FUNCTION F_TemperatureMethod : REAL
VAR_INPUT
	InputTemperature:	REAL;
END_VAR
VAR_OUTPUT
	Celsius : 		REAL;
	Fahrenheit : 	REAL;
	Kelvin : 		REAL;
	Cosine :		REAL;
END_VAR
VAR
	K: REAL;
	C: REAL;
	F: REAL;
END_VAR

// Function handling analog temperature measurement 
C := InputTemperature/10; 
K := C + 273.15;
F := C * 1.8 +32;

Cosine		 	:= COS(C);
Celsius 		:= C;
Fahrenheit 		:= F;
Kelvin 			:= K;

END_FUNCTION

(* stored: Version 1.1.0.1, ProductVersion 3.1.4024.10
   POU F_TemperatureMethod: Id {263ee18c-b0ce-433b-8548-28f5957fbdb5}, SpecialFunc None *)
